// TIA Portal V20 export
TYPE "UDT_Informe_DatosUT"
   STRUCT
      MesaDestino : UInt;
      TipoCarga : UInt;
      Enfradado : UInt;
      Flejado : UInt;
      Etiquetado : UInt;
      CotaAltura : UInt;
      CotaAnchura : UInt;
      CotaLargura : UInt;
      Peso : UDInt;
      AtributosCarga : Struct
         Vacia : Bool;
         Pila : Bool;
         Remontada : Bool;
      END_STRUCT;
      PosEtiqueta : Struct
         Derecha : Bool;
         Izquierda : Bool;
      END_STRUCT;
      etiqueta : Array[0..42] of Char;
      EtiquetaRouter : UDInt;
   END_STRUCT;
END_TYPE
